Xinje XDPPro project, PLC1: XD3-24 (software 3.5.3 2019-03-26 patch 3)

PROGRAM Ladder

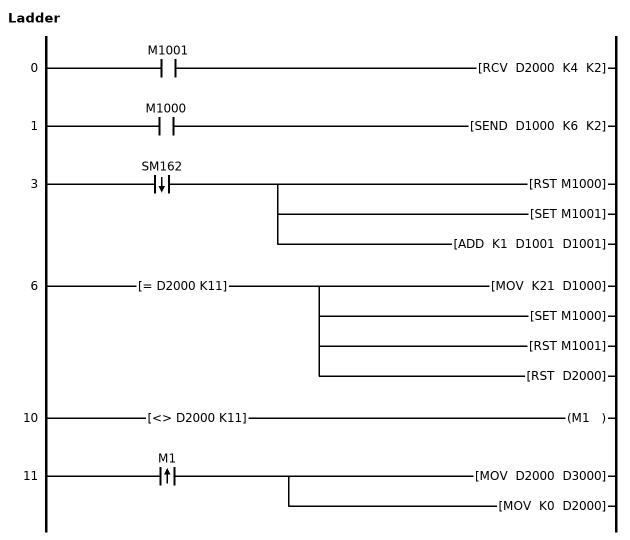
LD     M1001
RCV    D2000 K4 K2
LD     M1000
SEND   D1000 K6 K2
LDF    SM162
RST    M1000
SET    M1001
ADD    K1 D1001 D1001
LD=    D2000 K11
MOV    K21 D1000
SET    M1000
RST    M1001
RST    D2000
LD<>   D2000 K11
OUT    M1
LDP    M1
MOV    D2000 D3000
MOV    K0 D2000